// TIA Portal V18 export
DATA_BLOCK "AHUAO"   // DB112
{ S7_Optimized_Access := 'FALSE' }
VERSION : 0.1
// stored: AutoNumber false, DBAccessibleFromOPCUA true, IsOnlyStoredInLoadMemory false, IsWriteProtectedInAS false
   VAR
      AO { S7_SetPoint := 'True'} : "UTD_AHUsAO";
   END_VAR
BEGIN
END_DATA_BLOCK
